FUNCTION_BLOCK TEST_LWORD (* Test LWORD AND,OR,XOR *)
  (* Standard: 61131-3 *)
  (* Version 0.0, 2006-09-02, JHC, Holobloc Inc, Converted from TEST_BYTE. *)
  (* Compiler header: package fb.rt.test; *)
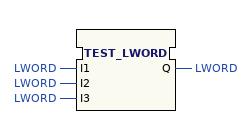
  VAR_INPUT
    I1 : LWORD;
    I2 : LWORD;
    I3 : LWORD;
  END_VAR
  VAR_OUTPUT
    Q : LWORD;
  END_VAR
  ALGORITHM REQ IN FBD:
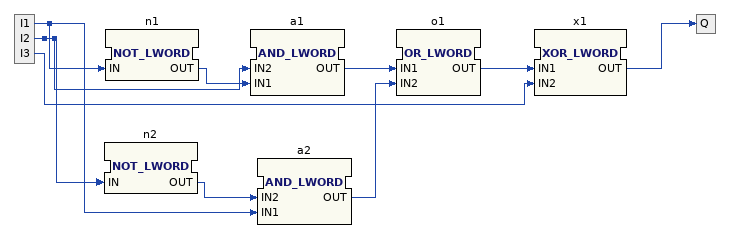
    FBS
      n1 : NOT_LWORD;
      n2 : NOT_LWORD;
      a1 : AND_LWORD;
      a2 : AND_LWORD;
      o1 : OR_LWORD;
      x1 : XOR_LWORD;
    END_FBS
    DATA_CONNECTIONS
      I1 TO n1.IN;
      I2 TO n2.IN;
      I2 TO a1.IN2;
      n2.OUT TO a2.IN2;
      n1.OUT TO a1.IN1;
      I1 TO a2.IN1;
      a1.OUT TO o1.IN1;
      a2.OUT TO o1.IN2;
      o1.OUT TO x1.IN1;
      I3 TO x1.IN2;
      x1.OUT TO Q;
    END_CONNECTIONS
  END_ALGORITHM
END_FUNCTION_BLOCK
